PROGRAM POUexecute
VAR
	iCount:INT;
	
	t1: TON;
	output: BOOL;
	e1: TIME;
	in1: BOOL;
	a: BOOL;
	b: BOOL;
	c: BOOL;
	out1: BOOL;
	t2: TON;
	out2: INT;
END_VAR

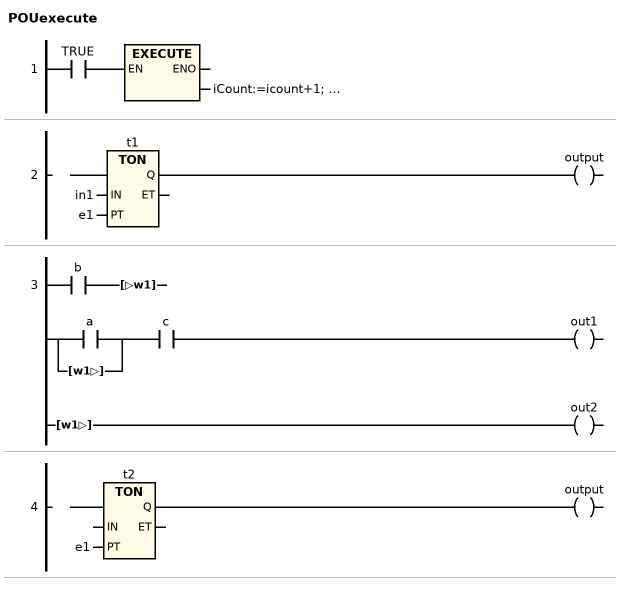
// NETWORK 1
iCount:=icount+1;

// NETWORK 2
t1(IN := in1, PT := e1); // TON
output := t1.Q;

// NETWORK 3
out1 := (a OR b) AND c;
out2 := b;

// NETWORK 4
t2(PT := e1); // TON
output := t2.Q;

END_PROGRAM

(* stored: Version 1.1.0.1, ProductVersion 3.1.4024.16
   POU POUexecute: Id {990f205a-b44a-4eb8-adf4-ef51ee7fa411}, SpecialFunc None *)
